FUNCTION Camera_Set_Ouput_Layout : UINT
VAR_INPUT
END_VAR
VAR
END_VAR

END_FUNCTION

(* stored: Version 1.1.0.1, ProductVersion 3.1.4024.10
   POU Camera_Set_Ouput_Layout: Id {f5de775a-8f45-4d98-a894-f355d5c529da}, SpecialFunc None *)
